IF THIS^.Step(996,TRUE,'Step number 996') THEN		
	THIS^.StepCompleteWhen((_RunOneStep OR _RunAllSteps) AND _FinishStep);	
	IF _RunOneStep THEN	
		_RunOneStep := FALSE;
		RETURN;
	END_IF	
END_IF		
		
IF THIS^.Step(997,TRUE,'Step number 997') THEN		
	THIS^.StepCompleteWhen((_RunOneStep OR _RunAllSteps) AND _FinishStep);	
	IF _RunOneStep THEN	
		_RunOneStep := FALSE;
		RETURN;
	END_IF	
END_IF		
		
IF THIS^.Step(998,TRUE,'Step number 998') THEN		
	THIS^.StepCompleteWhen((_RunOneStep OR _RunAllSteps) AND _FinishStep);	
	IF _RunOneStep THEN	
		_RunOneStep := FALSE;
		RETURN;
	END_IF	
END_IF		
		
IF THIS^.Step(999,TRUE,'Step number 999') THEN		
	THIS^.StepCompleteWhen((_RunOneStep OR _RunAllSteps) AND _FinishStep);	
	IF _RunOneStep THEN	
		_RunOneStep := FALSE;
		RETURN;
	END_IF	
END_IF		
		
IF THIS^.Step(1000,TRUE,'Step number 1000') THEN		
	THIS^.StepCompleteWhen((_RunOneStep OR _RunAllSteps) AND _FinishStep);	
	IF _RunOneStep THEN	
		_RunOneStep := FALSE;
		RETURN;
	END_IF	
END_IF		
		
IF THIS^.Step(1001,TRUE,'Step number 1001') THEN		
	THIS^.StepCompleteWhen((_RunOneStep OR _RunAllSteps) AND _FinishStep);	
	IF _RunOneStep THEN	
		_RunOneStep := FALSE;
		RETURN;
	END_IF	
END_IF		
		
IF THIS^.Step(1002,TRUE,'Step number 1002') THEN		
	THIS^.StepCompleteWhen((_RunOneStep OR _RunAllSteps) AND _FinishStep);	
	IF _RunOneStep THEN	
		_RunOneStep := FALSE;
		RETURN;
	END_IF	
END_IF		
		
IF THIS^.Step(1003,TRUE,'Step number 1003') THEN		
	THIS^.StepCompleteWhen((_RunOneStep OR _RunAllSteps) AND _FinishStep);	
	IF _RunOneStep THEN	
		_RunOneStep := FALSE;
		RETURN;
	END_IF	
END_IF		
		
IF THIS^.Step(1004,TRUE,'Step number 1004') THEN		
	THIS^.StepCompleteWhen((_RunOneStep OR _RunAllSteps) AND _FinishStep);	
	IF _RunOneStep THEN	
		_RunOneStep := FALSE;
		RETURN;
	END_IF	
END_IF		
		
IF THIS^.Step(1005,TRUE,'Step number 1005') THEN		
	THIS^.StepCompleteWhen((_RunOneStep OR _RunAllSteps) AND _FinishStep);	
	IF _RunOneStep THEN	
		_RunOneStep := FALSE;
		RETURN;
	END_IF	
END_IF		
		
IF THIS^.Step(1006,TRUE,'Step number 1006') THEN		
	THIS^.StepCompleteWhen((_RunOneStep OR _RunAllSteps) AND _FinishStep);	
	IF _RunOneStep THEN	
		_RunOneStep := FALSE;
		RETURN;
	END_IF	
END_IF		
		
IF THIS^.Step(1007,TRUE,'Step number 1007') THEN		
	THIS^.StepCompleteWhen((_RunOneStep OR _RunAllSteps) AND _FinishStep);	
	IF _RunOneStep THEN	
		_RunOneStep := FALSE;
		RETURN;
	END_IF	
END_IF		
		
IF THIS^.Step(1008,TRUE,'Step number 1008') THEN		
	THIS^.StepCompleteWhen((_RunOneStep OR _RunAllSteps) AND _FinishStep);	
	IF _RunOneStep THEN	
		_RunOneStep := FALSE;
		RETURN;
	END_IF	
END_IF		
		
IF THIS^.Step(1009,TRUE,'Step number 1009') THEN		
	THIS^.StepCompleteWhen((_RunOneStep OR _RunAllSteps) AND _FinishStep);	
	IF _RunOneStep THEN	
		_RunOneStep := FALSE;
		RETURN;
	END_IF	
END_IF		
		
IF THIS^.Step(1010,TRUE,'Step number 1010') THEN		
	THIS^.StepCompleteWhen((_RunOneStep OR _RunAllSteps) AND _FinishStep);	
	IF _RunOneStep THEN	
		_RunOneStep := FALSE;
		RETURN;
	END_IF	
END_IF		
		
IF THIS^.Step(1011,TRUE,'Step number 1011') THEN		
	THIS^.StepCompleteWhen((_RunOneStep OR _RunAllSteps) AND _FinishStep);	
	IF _RunOneStep THEN	
		_RunOneStep := FALSE;
		RETURN;
	END_IF	
END_IF		
		
IF THIS^.Step(1012,TRUE,'Step number 1012') THEN		
	THIS^.StepCompleteWhen((_RunOneStep OR _RunAllSteps) AND _FinishStep);	
	IF _RunOneStep THEN	
		_RunOneStep := FALSE;
		RETURN;
	END_IF	
END_IF		
		
IF THIS^.Step(1013,TRUE,'Step number 1013') THEN		
	THIS^.StepCompleteWhen((_RunOneStep OR _RunAllSteps) AND _FinishStep);	
	IF _RunOneStep THEN	
		_RunOneStep := FALSE;
		RETURN;
	END_IF	
END_IF		
		
IF THIS^.Step(1014,TRUE,'Step number 1014') THEN		
	THIS^.StepCompleteWhen((_RunOneStep OR _RunAllSteps) AND _FinishStep);	
	IF _RunOneStep THEN	
		_RunOneStep := FALSE;
		RETURN;
	END_IF	
END_IF		
		
IF THIS^.Step(1015,TRUE,'Step number 1015') THEN		
	THIS^.StepCompleteWhen((_RunOneStep OR _RunAllSteps) AND _FinishStep);	
	IF _RunOneStep THEN	
		_RunOneStep := FALSE;
		RETURN;
	END_IF	
END_IF		
		
IF THIS^.Step(1016,TRUE,'Step number 1016') THEN		
	THIS^.StepCompleteWhen((_RunOneStep OR _RunAllSteps) AND _FinishStep);	
	IF _RunOneStep THEN	
		_RunOneStep := FALSE;
		RETURN;
	END_IF	
END_IF		
		
IF THIS^.Step(1017,TRUE,'Step number 1017') THEN		
	THIS^.StepCompleteWhen((_RunOneStep OR _RunAllSteps) AND _FinishStep);	
	IF _RunOneStep THEN	
		_RunOneStep := FALSE;
		RETURN;
	END_IF	
END_IF		
		
IF THIS^.Step(1018,TRUE,'Step number 1018') THEN		
	THIS^.StepCompleteWhen((_RunOneStep OR _RunAllSteps) AND _FinishStep);	
	IF _RunOneStep THEN	
		_RunOneStep := FALSE;
		RETURN;
	END_IF	
END_IF		
		
IF THIS^.Step(1019,TRUE,'Step number 1019') THEN		
	THIS^.StepCompleteWhen((_RunOneStep OR _RunAllSteps) AND _FinishStep);	
	IF _RunOneStep THEN	
		_RunOneStep := FALSE;
		RETURN;
	END_IF	
END_IF		
		
IF THIS^.Step(1020,TRUE,'Step number 1020') THEN		
	THIS^.StepCompleteWhen((_RunOneStep OR _RunAllSteps) AND _FinishStep);	
	IF _RunOneStep THEN	
		_RunOneStep := FALSE;
		RETURN;
	END_IF	
END_IF		
		
IF THIS^.Step(1021,TRUE,'Step number 1021') THEN		
	THIS^.StepCompleteWhen((_RunOneStep OR _RunAllSteps) AND _FinishStep);	
	IF _RunOneStep THEN	
		_RunOneStep := FALSE;
		RETURN;
	END_IF	
END_IF		
		
IF THIS^.Step(1022,TRUE,'Step number 1022') THEN		
	THIS^.StepCompleteWhen((_RunOneStep OR _RunAllSteps) AND _FinishStep);	
	IF _RunOneStep THEN	
		_RunOneStep := FALSE;
		RETURN;
	END_IF	
END_IF		
		
IF THIS^.Step(1023,TRUE,'Step number 1023') THEN		
	THIS^.StepCompleteWhen((_RunOneStep OR _RunAllSteps) AND _FinishStep);	
	IF _RunOneStep THEN	
		_RunOneStep := FALSE;
		RETURN;
	END_IF	
END_IF		
		
//******************************************************************
IF THIS^.Step(_ID,_Enabled,_StepDescription) THEN
	THIS^.StepCompleteWhen((_RunOneStep OR _RunAllSteps) AND _FinishStep);	
	IF _RunOneStep THEN	
		_RunOneStep := FALSE;
		RETURN;
	END_IF		
END_IF
END_METHOD

METHOD PUBLIC PostSequenceComplete
_PostSequenceCompleteCount := _PostSequenceCompleteCount + 1;
END_METHOD

METHOD PUBLIC PostStepComplete
_PostStepCompleteCount := _PostStepCompleteCount + 1;
END_METHOD

PROPERTY INTERNAL RequestStepCycle : UINT
GET
RequestStepCycle := _requestStepCycle;
END_GET
SET
_requestStepCycle := RequestStepCycle;
END_SET
END_PROPERTY

METHOD SequencerClose
SUPER^.Close();
END_METHOD

METHOD INTERNAL SequencerHasError : BOOL
SequencerHasError := SUPER^._sequencerHasError;
END_METHOD

METHOD SequencerOpen
SUPER^.Open();
END_METHOD

METHOD INTERNAL SetChildState 
VAR_INPUT
	inState			:	INT;
END_VAR
THIS^._TcoState.ChangeState(inState);
END_METHOD

METHOD INTERNAL SetCurrentStep 
VAR_INPUT
	inStepID 			:	INT;
	inStepDescription	:	STRING(254);
END_VAR
THIS^._currentStep.ID			:=	inStepID;
THIS^._currentStep.Description	:=	inStepDescription;
END_METHOD

METHOD INTERNAL SetNumberOfSteps 
VAR_INPUT
	inNumberOfSteps : UINT;
END_VAR
_stepCounter 						:=	inNumberOfSteps;
_numberOfStepsInSequence			:=	inNumberOfSteps;
_previousNumberOfStepsInSequence 	:=	inNumberOfSteps;
END_METHOD

METHOD INTERNAL SetSequenceAsChecked
_stepIDUniquenessChecked := TRUE;
END_METHOD

METHOD INTERNAL SetSequenceAsNotChecked
_stepIDUniquenessChecked := FALSE;
END_METHOD

METHOD INTERNAL SetTestParams
VAR_INPUT
	inRunOneStep		:	BOOL;
	inRunAllSteps		:	BOOL;
	inFinishStep		:	BOOL;
	inID				:	UINT;
	inEnabled			:	BOOL;
	inStepDescription	:	STRING(254);	
END_VAR
THIS^._RunOneStep		:=			inRunOneStep;
THIS^._RunAllSteps 		:= 			inRunAllSteps;
THIS^._FinishStep 		:= 			inFinishStep;
THIS^._ID 				:=			inID;
THIS^._Enabled 			:= 			inEnabled;
THIS^._StepDescription 	:=			inStepDescription;
END_METHOD

METHOD INTERNAL UpdateCurrentStepDetails
_currentStepId				:=	SUPER^._currentStep.ID;
_currentStepOrder			:=	SUPER^._currentStep.Order;
_currentStepEnabled			:=	SUPER^._currentStep.Enabled;
_currentStepDescription		:=	SUPER^._currentStep.Description;
_currentStepStatus			:=	SUPER^._currentStep.Status;
_currentStepDuration		:=	SUPER^._currentStep.Duration;
END_METHOD

END_FUNCTION_BLOCK

(* stored: Version 1.1.0.1, ProductVersion 3.1.4024.6
   POU _TcoSequencer: Id {ac19fe4f-0c0e-08e9-3df5-0840192e4ee2}, SpecialFunc None
   Folder _Tests: Id {36ff3928-274d-02d5-18e6-23dcd25a0584}
   Method ChildHasAutoRestoreEnabled: Id {2fe344f3-4fea-0846-0ec8-378fe51cb4c6}
   Method ChildIsAutoRestorable: Id {e0cb2365-b187-0b05-2101-33f128967786}
   Method CleanupPointers: Id {c754833e-788e-0dc0-39b2-57f91228c555}
   Method ClearNumberOfSteps: Id {ccb8339d-f888-01c2-334c-f78620010950}
   Method GetChildState: Id {aaac1bd4-eac0-002e-3f58-ea6c5e49e949}
   Method GetSequencerErrorId: Id {cfa5c7b8-bdaa-0dc9-318b-07d87a737808}
   Method GetTextOfTheMostImportantMessage: Id {0f5e0607-86a0-04f2-3053-f70b778527fb}
   Method HasAutoRestoreEnabled: Id {13163512-5f77-0a1f-15bd-0485ab98dc6e}
   Method IsAutoRestorable: Id {78b773c3-e01b-01ec-3871-0a0bdbd810d6}
   Method IsFirstStepEntry: Id {4f006540-c701-07be-1eb3-95b9c8a360ee}
   Method Main: Id {3a6cbc53-5690-0480-174f-e4140d338a45}
   Method PostSequenceComplete: Id {2fd78922-07d4-01ec-1736-1c3b4b7d9bd8}
   Method PostStepComplete: Id {154d4f23-050b-01f6-08b9-2a631c3ec621}
   Property RequestStepCycle: Id {c2da0157-c6b1-052f-064f-3e3f6d17de69}
   Get Get: Id {6b43bca9-2a6f-0436-073d-241b14a17d9a}
   Set Set: Id {66bd96b6-e8a3-0fe0-344b-3b831339bba2}
   Method SequencerClose: Id {f3addcb4-0fda-0a2d-0925-430c6f4ad3f8}
   Method SequencerHasError: Id {07e19515-04c8-048f-12a4-f42415093577}
   Method SequencerOpen: Id {b4334737-6cb3-0eba-0d2f-cd067be7b53d}
   Method SetChildState: Id {60024768-516f-0fd2-2f16-e270836f2db6}
   Method SetCurrentStep: Id {223d2a4f-ee82-0c54-0227-548f61243f4d}
   Method SetNumberOfSteps: Id {a8a0d4fb-e225-0fb8-3c9b-d2a796c1b2ec}
   Method SetSequenceAsChecked: Id {43e68eca-b921-0c50-2ca5-03882ac05b27}
   Method SetSequenceAsNotChecked: Id {09a6a7e6-7763-040e-016a-fc5c2ce30618}
   Method SetTestParams: Id {7a624c26-ee8b-0b24-15f9-09fad6ccc521}
   Method UpdateCurrentStepDetails: Id {590d6a94-7182-0c50-1bd0-bf34e87df18c} *)
